// TIA Portal V16 export
// export: Created 2022-02-04T14:40:10.1877338Z, ExportSetting WithDefaults, DisplayName Totally Integrated Automation Portal, DisplayVersion V16 Update 1, DisplayName TIA Portal Version Control Interface, DisplayVersion V16, DisplayName TIA Portal Openness, DisplayVersion V16, DisplayName SINAMICS Startdrive Advanced, DisplayVersion V16 Update 5, DisplayName SINAMICS Startdrive G130, G150, S120, S150, SINAMICS MV, S210, DisplayVersion V16 Update 5, DisplayName SINAMICS Startdrive G110M, G120, G120C, G120D, G120P, G115D, DisplayVersion V16 Update 5, DisplayName STEP 7 Professional, DisplayVersion V16, DisplayName STEP 7 Safety, DisplayVersion V16, DisplayName WinCC Advanced, DisplayVersion V16, DisplayName SIMATIC Visualization Architect, DisplayVersion V16
FUNCTION_BLOCK "Загрузка"   // FB8, LAD
VERSION : 0.1
// stored: AutoNumber true, IsIECCheckEnabled false, UDAEnableTagReadback false
   VAR DB_SPECIFIC
      "TrigS84.4" : Bool;
      LiftUpTrig : Bool;
      "212StartCNTL" : Bool;
      "TrigS82.3/S76.5" : Bool;
      LiftDownTrig : Bool;
   END_VAR
   VAR_TEMP
      Sert : Word;
      AutoLamp : Bool;
      M213_wide_mode : Bool;
   END_VAR
   VAR_TEMP   // added for the SCL form of the ladder/FBD networks
      _w1 : Bool;
      _s5time1 : S5Time;
      _w2 : Bool;
      _w3 : Bool;
      _w4 : Bool;
      _s5time2 : S5Time;
   END_VAR
BEGIN

REGION Network 1: 211 группа на 4 мотора обющий сигнал готовности
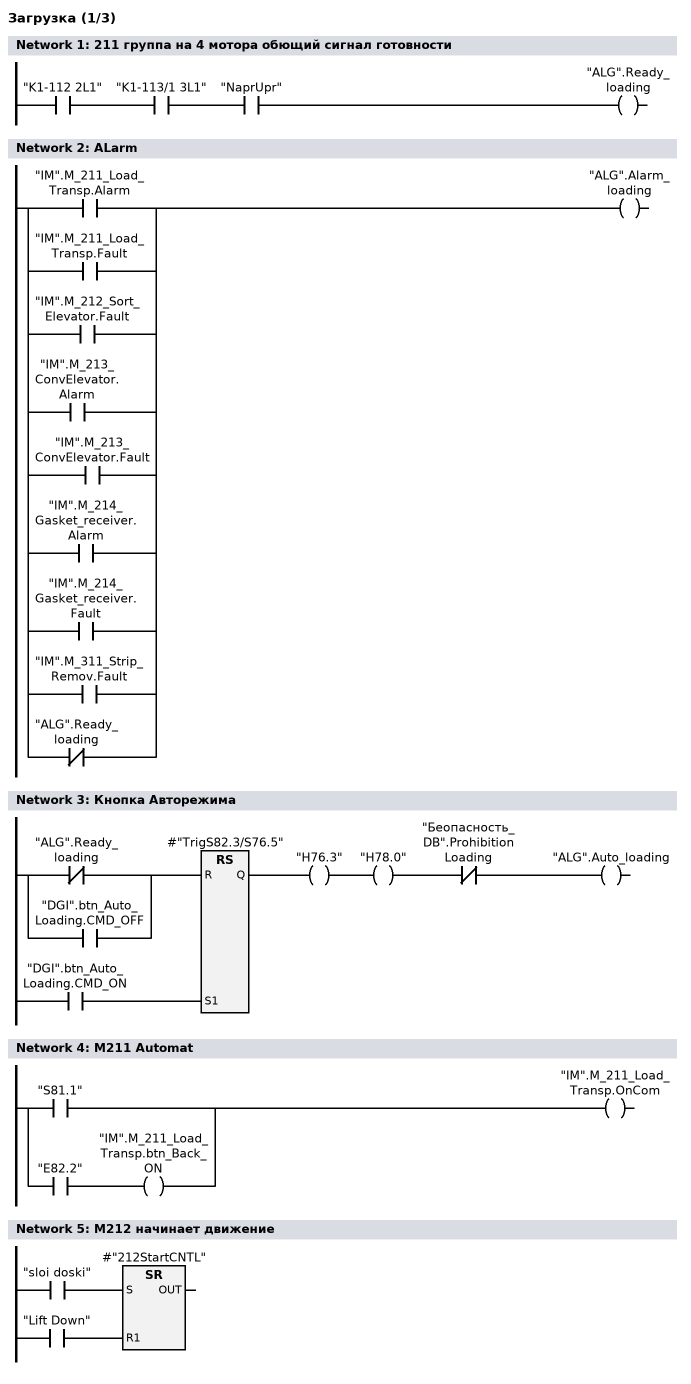
   RUNG wire#powerrail
      Contact( "K1-112 2L1" )
      Contact( "K1-113/1 3L1" )
      Contact( "NaprUpr" )
      Coil( "ALG".Ready_loading )
   END_RUNG
   // the same network as SCL:
   "ALG".Ready_loading := "K1-112 2L1" AND "K1-113/1 3L1" AND "NaprUpr";
END_REGION

REGION Network 2: ALarm
   RUNG wire#powerrail
      Contact( "IM".M_211_Load_Transp.Alarm )
      wire#w1
      Coil( "ALG".Alarm_loading )
   END_RUNG
   RUNG wire#powerrail
      Contact( "IM".M_211_Load_Transp.Fault )
   END_RUNG wire#w1
   RUNG wire#powerrail
      Contact( "IM".M_212_Sort_Elevator.Fault )
   END_RUNG wire#w1
   RUNG wire#powerrail
      Contact( "IM".M_213_ConvElevator.Alarm )
   END_RUNG wire#w1
   RUNG wire#powerrail
      Contact( "IM".M_213_ConvElevator.Fault )
   END_RUNG wire#w1
   RUNG wire#powerrail
      Contact( "IM".M_214_Gasket_receiver.Alarm )
   END_RUNG wire#w1
   RUNG wire#powerrail
      Contact( "IM".M_214_Gasket_receiver.Fault )
   END_RUNG wire#w1
   RUNG wire#powerrail
      Contact( "IM".M_311_Strip_Remov.Fault )
   END_RUNG wire#w1
   RUNG wire#powerrail
      I_Contact( "ALG".Ready_loading )
   END_RUNG wire#w1
   // the same network as SCL:
   "ALG".Alarm_loading := "IM".M_211_Load_Transp.Alarm OR "IM".M_211_Load_Transp.Fault OR "IM".M_212_Sort_Elevator.Fault OR "IM".M_213_ConvElevator.Alarm OR "IM".M_213_ConvElevator.Fault OR "IM".M_214_Gasket_receiver.Alarm OR "IM".M_214_Gasket_receiver.Fault OR "IM".M_311_Strip_Remov.Fault OR NOT "ALG".Ready_loading;
END_REGION

REGION Network 3: Кнопка Авторежима
   RUNG wire#powerrail
      I_Contact( "ALG".Ready_loading )
      wire#w1
      S_RS(operand := #"TrigS82.3/S76.5", s1 := wire#w2)
      Coil( "H76.3" )
      Coil( "H78.0" )
      I_Contact( "Беопасность_DB".ProhibitionLoading )
      Coil( "ALG".Auto_loading )
   END_RUNG
   RUNG wire#powerrail
      Contact( "DGI".btn_Auto_Loading.CMD_OFF )
   END_RUNG wire#w1
   RUNG wire#powerrail
      Contact( "DGI".btn_Auto_Loading.CMD_ON )
   END_RUNG wire#w2
   // the same network as SCL:
   IF NOT "ALG".Ready_loading OR "DGI".btn_Auto_Loading.CMD_OFF THEN
       #"TrigS82.3/S76.5" := FALSE;   // RS flip-flop
   END_IF;
   IF "DGI".btn_Auto_Loading.CMD_ON THEN #"TrigS82.3/S76.5" := TRUE; END_IF;
   "H76.3" := #"TrigS82.3/S76.5";
   "H78.0" := #"TrigS82.3/S76.5";
   "ALG".Auto_loading := #"TrigS82.3/S76.5" AND NOT "Беопасность_DB".ProhibitionLoading;
END_REGION

REGION Network 4: M211 Automat
   RUNG wire#powerrail
      Contact( "S81.1" )
      wire#w1
      Coil( "IM".M_211_Load_Transp.OnCom )
   END_RUNG
   RUNG wire#powerrail
      Contact( "E82.2" )
      Coil( "IM".M_211_Load_Transp.btn_Back_ON )
   END_RUNG wire#w1
   // the same network as SCL:
   "IM".M_211_Load_Transp.btn_Back_ON := "E82.2";
   "IM".M_211_Load_Transp.OnCom := "S81.1" OR "E82.2";
END_REGION

REGION Network 5: M212 начинает движение
   RUNG wire#powerrail
      Contact( "sloi doski" )
      S_SR(operand := #"212StartCNTL", r1 := wire#w1)
   END_RUNG
   RUNG wire#powerrail
      Contact( "Lift Down" )
   END_RUNG wire#w1
   // the same network as SCL:
   IF "sloi doski" THEN
       #"212StartCNTL" := TRUE;   // SR flip-flop
   END_IF;
   IF "Lift Down" THEN #"212StartCNTL" := FALSE; END_IF;
END_REGION

REGION Network 6: М212 AutoMode
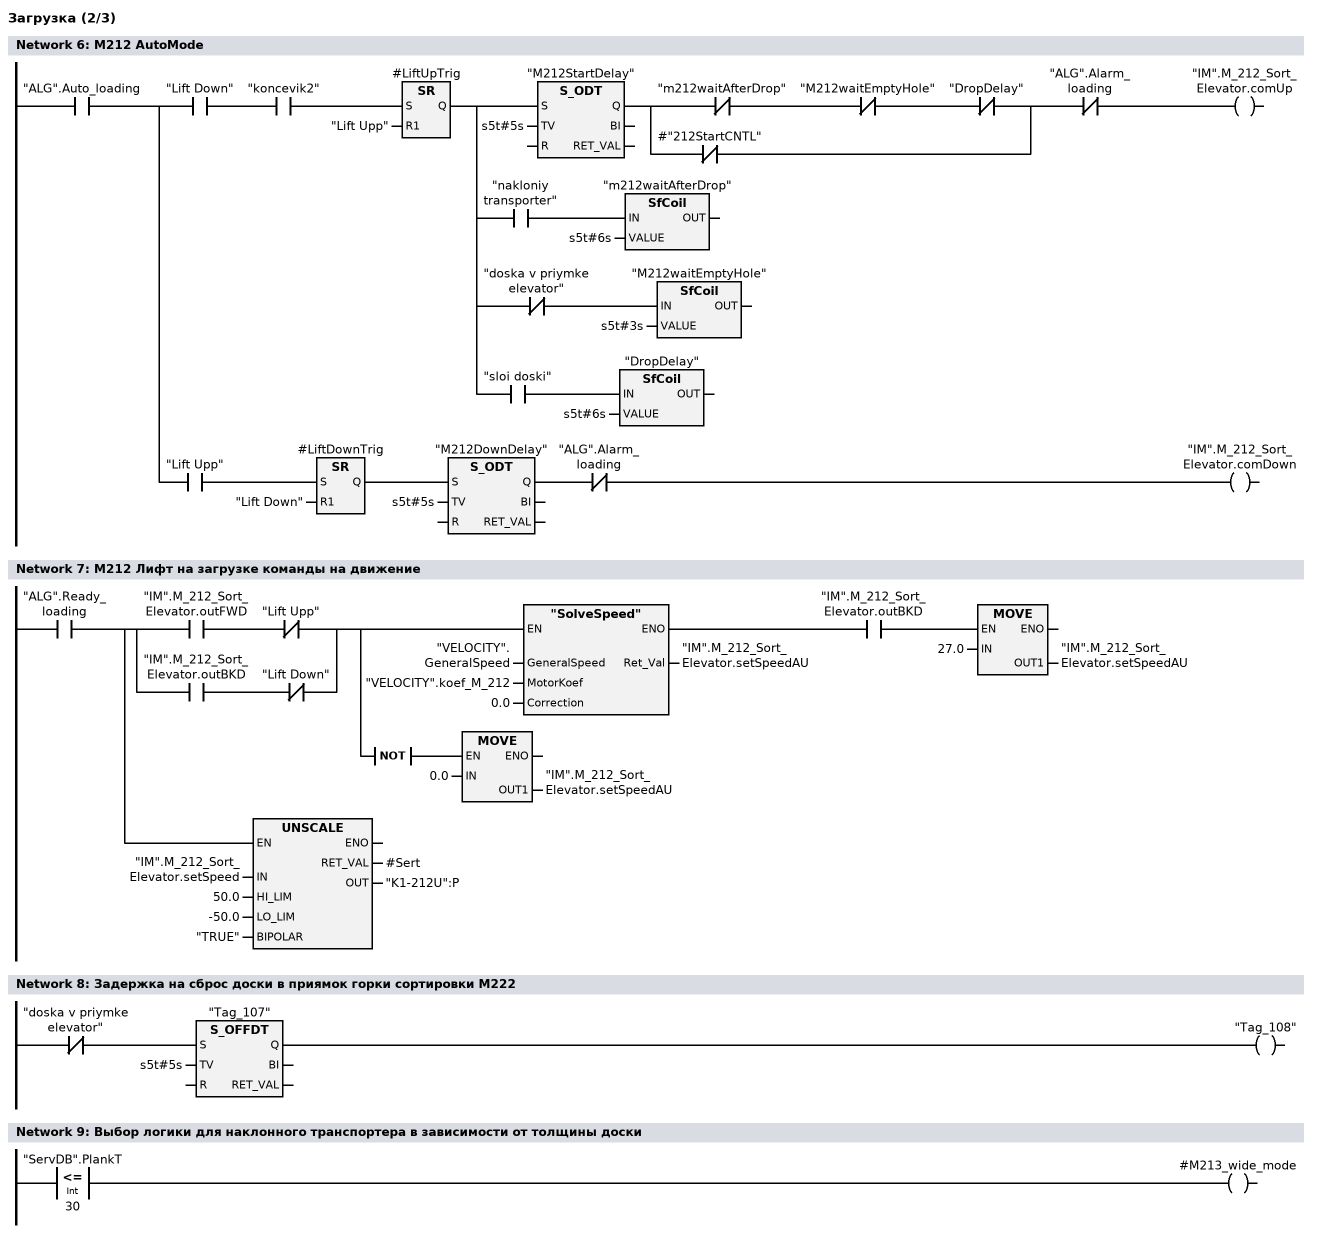
   // no SCL statement known for SfCoil: written as a call
   IF "ALG".Auto_loading AND "Lift Down" AND "koncevik2" THEN
       #LiftUpTrig := TRUE;   // SR flip-flop
   END_IF;
   IF "Lift Upp" THEN #LiftUpTrig := FALSE; END_IF;
   #_w2 := #LiftUpTrig;
   #_s5time1 := S_ODT(T_NO := "M212StartDelay", S := #LiftUpTrig, TV := s5t#5s, Q => #_w1);
   "IM".M_212_Sort_Elevator.comUp := #_w1 AND ((NOT "m212waitAfterDrop" AND NOT "M212waitEmptyHole" AND NOT "DropDelay") OR NOT #"212StartCNTL") AND NOT "ALG".Alarm_loading;
   #_w3 := "ALG".Auto_loading;
   SfCoil(in := #_w2 AND "nakloniy transporter", value := s5t#6s, operand := "m212waitAfterDrop");
   SfCoil(in := #_w2 AND NOT "doska v priymke elevator", value := s5t#3s, operand := "M212waitEmptyHole");
   SfCoil(in := #_w2 AND "sloi doski", value := s5t#6s, operand := "DropDelay");
   IF #_w3 AND "Lift Upp" THEN
       #LiftDownTrig := TRUE;   // SR flip-flop
   END_IF;
   IF "Lift Down" THEN #LiftDownTrig := FALSE; END_IF;
   #_s5time2 := S_ODT(T_NO := "M212DownDelay", S := #LiftDownTrig, TV := s5t#5s, Q => #_w4);
   "IM".M_212_Sort_Elevator.comDown := #_w4 AND NOT "ALG".Alarm_loading;
END_REGION

REGION Network 7: М212 Лифт на загрузке команды на движение
   RUNG wire#powerrail
      Contact( "ALG".Ready_loading )
      wire#w1
      Contact( "IM".M_212_Sort_Elevator.outFWD )
      I_Contact( "Lift Upp" )
      wire#w2
      "SolveSpeed"(GeneralSpeed := "VELOCITY".GeneralSpeed, MotorKoef := "VELOCITY".koef_M_212, Correction := 0.0, Ret_Val => "IM".M_212_Sort_Elevator.setSpeedAU)
      Contact( "IM".M_212_Sort_Elevator.outBKD )
      { S7_GenerateENO := "TRUE" } Move(in := 27.0, out1 => "IM".M_212_Sort_Elevator.setSpeedAU)
   END_RUNG
   RUNG wire#w1
      Contact( "IM".M_212_Sort_Elevator.outBKD )
      I_Contact( "Lift Down" )
   END_RUNG wire#w2
   RUNG wire#w2
      Not()
      { S7_GenerateENO := "TRUE" } Move(in := 0.0, out1 => "IM".M_212_Sort_Elevator.setSpeedAU)
   END_RUNG
   RUNG wire#w1
      UNSCALE(IN := "IM".M_212_Sort_Elevator.setSpeed, HI_LIM := 50.0, LO_LIM := -50.0, BIPOLAR := "TRUE", RET_VAL => #Sert, OUT => "K1-212U":P)
   END_RUNG
   // the same network as SCL:
   #_w1 := "ALG".Ready_loading AND (("IM".M_212_Sort_Elevator.outFWD AND NOT "Lift Upp") OR ("IM".M_212_Sort_Elevator.outBKD AND NOT "Lift Down"));
   #_w3 := "ALG".Ready_loading;
   "IM".M_212_Sort_Elevator.setSpeedAU := "SolveSpeed"(EN := #_w1,
                           GeneralSpeed := "VELOCITY".GeneralSpeed,
                           MotorKoef := "VELOCITY".koef_M_212,
                           Correction := 0.0,
                           ENO => #_w2);
   IF #_w2 AND "IM".M_212_Sort_Elevator.outBKD THEN "IM".M_212_Sort_Elevator.setSpeedAU := 27.0; END_IF;
   IF NOT #_w1 THEN "IM".M_212_Sort_Elevator.setSpeedAU := 0.0; END_IF;
   IF #_w3 THEN
       #Sert := UNSCALE(IN := "IM".M_212_Sort_Elevator.setSpeed,
                        HI_LIM := 50.0,
                        LO_LIM := -50.0,
                        BIPOLAR := "TRUE",
                        OUT => "K1-212U":P);
   END_IF;
END_REGION

REGION Network 8: Задержка на сброс доски в приямок горки сортировки М222
   RUNG wire#powerrail
      I_Contact( "doska v priymke elevator" )
      S_OFFDT(T_NO := "Tag_107", TV := s5t#5s, R :=, BI =>, RET_VAL =>)
      Coil( "Tag_108" )
   END_RUNG
   // the same network as SCL:
   #_s5time1 := S_OFFDT(T_NO := "Tag_107", S := NOT "doska v priymke elevator", TV := s5t#5s, Q => #_w1);
   "Tag_108" := #_w1;
END_REGION

REGION Network 9: Выбор логики для наклонного транспортера в зависимости от толщины доски
   RUNG wire#powerrail
      { S7_Templates := "SrcType := Int" } LE_Contact(in1 := "ServDB".PlankT, in2 := 30)
      Coil( #M213_wide_mode )
   END_RUNG
   // the same network as SCL:
   #M213_wide_mode := "ServDB".PlankT <= 30;
END_REGION

REGION Network 10: М213 Наклонный транспортер Авто вперед
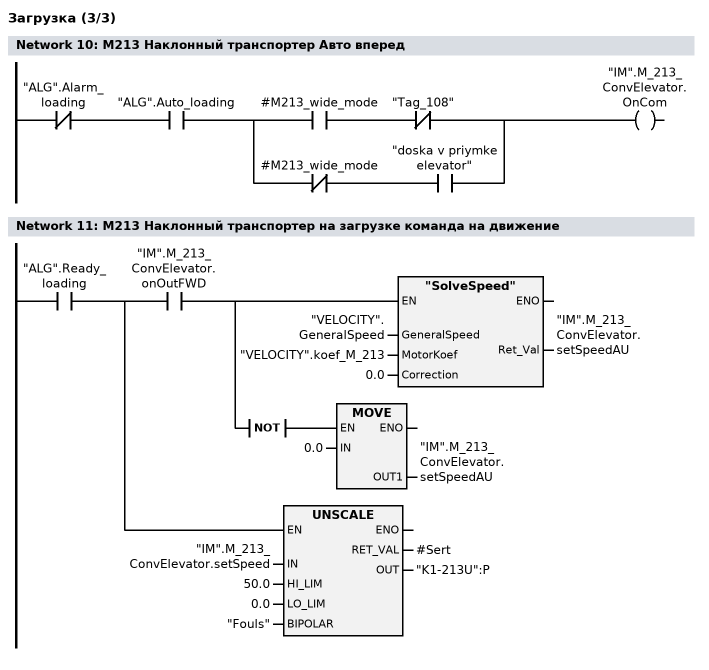
   RUNG wire#powerrail
      I_Contact( "ALG".Alarm_loading )
      Contact( "ALG".Auto_loading )
      wire#w1
      Contact( #M213_wide_mode )
      I_Contact( "Tag_108" )
      wire#w2
      Coil( "IM".M_213_ConvElevator.OnCom )
   END_RUNG
   RUNG wire#w1
      I_Contact( #M213_wide_mode )
      Contact( "doska v priymke elevator" )
   END_RUNG wire#w2
   // the same network as SCL:
   "IM".M_213_ConvElevator.OnCom := NOT "ALG".Alarm_loading AND "ALG".Auto_loading AND ((#M213_wide_mode AND NOT "Tag_108") OR (NOT #M213_wide_mode AND "doska v priymke elevator"));
END_REGION

REGION Network 11: М213 Наклонный транспортер на загрузке команда на движение
   RUNG wire#powerrail
      Contact( "ALG".Ready_loading )
      wire#w1
      Contact( "IM".M_213_ConvElevator.onOutFWD )
      wire#w2
      "SolveSpeed"(GeneralSpeed := "VELOCITY".GeneralSpeed, MotorKoef := "VELOCITY".koef_M_213, Correction := 0.0, Ret_Val => "IM".M_213_ConvElevator.setSpeedAU)
   END_RUNG
   RUNG wire#w2
      Not()
      { S7_GenerateENO := "TRUE" } Move(in := 0.0, out1 => "IM".M_213_ConvElevator.setSpeedAU)
   END_RUNG
   RUNG wire#w1
      UNSCALE(IN := "IM".M_213_ConvElevator.setSpeed, HI_LIM := 50.0, LO_LIM := 0.0, BIPOLAR := "Fouls", RET_VAL => #Sert, OUT => "K1-213U":P)
   END_RUNG
   // the same network as SCL:
   #_w1 := "ALG".Ready_loading AND "IM".M_213_ConvElevator.onOutFWD;
   #_w2 := "ALG".Ready_loading;
   IF #_w1 THEN
       "IM".M_213_ConvElevator.setSpeedAU := "SolveSpeed"(GeneralSpeed := "VELOCITY".GeneralSpeed,
                               MotorKoef := "VELOCITY".koef_M_213,
                               Correction := 0.0);
   END_IF;
   IF NOT #_w1 THEN "IM".M_213_ConvElevator.setSpeedAU := 0.0; END_IF;
   IF #_w2 THEN
       #Sert := UNSCALE(IN := "IM".M_213_ConvElevator.setSpeed,
                        HI_LIM := 50.0,
                        LO_LIM := 0.0,
                        BIPOLAR := "Fouls",
                        OUT => "K1-213U":P);
   END_IF;
END_REGION
END_FUNCTION_BLOCK
